// SIMATIC S7-200 project (STEP 7-Micro/WIN), CPU 224 REL 02.01

SYMBOL_TABLE USER1
lightSensor      V0.0
openDoor         V0.1
lowBob           V0.2
upBob            V0.3
heaterGoOn       V2.0
lightGoOn        V2.1
doorGoOpen       V2.2
ventilGoOn       V2.3
valve1goOn       V2.4
valve2goOn       V2.5
valve3goOn       V2.6
lightBySensor    V3.0
lightByTime      V3.1
lightHandOn      V3.2
lightHandOff     V3.3
heatSensorIsAir  V3.4
heatHandOn       V3.5
heatHandOff      V3.6
doorHandOn       V3.7
doorHandOff      V4.0
setClock         V4.1
readYear         VB50
readMonth        VB51
readDay          VB52
readHours        VB53
readMinutes      VB54
readSeconds      VB55
readWeekday      VB57
writeYear        VB58
writeMonth       VB59
writeDay         VB60
writeHours       VB61
writeMinutes     VB62
writeSeconds     VB63
writeWeekday     VB65
v1_e1_on_hh      VB148
v1_e1_on_mm      VB149
v1_e1_off_hh     VB150
v1_e1_off_mm     VB151
v1_e2_on_hh      VB152
v1_e2_on_mm      VB153
v1_e2_off_hh     VB154
v1_e2_off_mm     VB155
v1_e3_on_hh      VB156
v1_e3_on_mm      VB157
v1_e3_off_hh     VB158
v1_e3_off_mm     VB159
v1_e4_on_hh      VB160
v1_e4_on_mm      VB161
v1_e4_off_hh     VB162
v1_e4_off_mm     VB163
v1_e5_on_hh      VB164
v1_e5_on_mm      VB165
v1_e5_off_hh     VB166
v1_e5_off_mm     VB167
v2_e1_on_hh      VB168
v2_e1_on_mm      VB169
v2_e1_off_hh     VB170
v2_e1_off_mm     VB171
v2_e2_on_hh      VB172
v2_e2_on_mm      VB173
v2_e2_off_hh     VB174
v2_e2_off_mm     VB175
v2_e3_on_hh      VB176
v2_e3_on_mm      VB177
v2_e3_off_hh     VB178
v2_e3_off_mm     VB179
v2_e4_on_hh      VB180
v2_e4_on_mm      VB181
v2_e4_off_hh     VB182
v2_e4_off_mm     VB183
v2_e5_on_hh      VB184
v2_e5_on_mm      VB185
v2_e5_off_hh     VB186
v2_e5_off_mm     VB187
light_e1_on_hh   VB188
light_e1_on_mm   VB189
light_e1_off_hh  VB190
light_e1_off_mm  VB191
light_e2_on_hh   VB192
light_e2_on_mm   VB193
light_e2_off_hh  VB194
light_e2_off_mm  VB195
door_e1_on_hh    VB212
door_e1_on_mm    VB213
door_e1_off_hh   VB214
door_e1_off_mm   VB215
door_e2_on_hh    VB216
door_e2_on_mm    VB217
door_e2_off_hh   VB218
door_e2_off_mm   VB219
roomTemp4ma      VD100
roomTemp20ma     VD104
airTemp4ma       VD108
airTemp20ma      VD112
humidityRoom4ma  VD116
humidityRoom20ma VD120
floorTemp4ma     VD124
floorTemp20ma    VD128
roomTemp         VD132
airTemp          VD136
humidityRoom     VD140
floorTemp        VD144
lowSpWithAir     VD196
upSpWithAir      VD200
lowSpWithFloor   VD204
upSpWithFloor    VD208
lightTimeGo      V4.2
doorTimeGo       V4.3
heatTempGo       V4.4
lightHandGo      V4.5
doorHandGo       V4.6
heatHandGo       V4.7
ventilSensorIsTemp V5.0
lowSpWithTemp    VD220
upSpWithTemp     VD224
lowSpWithHumi    VD228
upSpWithHumi     VD232
lowSpWithOutside VD236
upSpWithOutside  VD240
heat2goOn        V5.1
im1_e1_on_hh     VB244
im1_e1_on_mm     VB245
im1_e1_off_hh    VB246
im1_e1_off_mm    VB247
im1_e2_on_hh     VB248
im1_e2_on_mm     VB249
im1_e2_off_hh    VB250
im1_e2_off_mm    VB251
im1_e3_on_hh     VB252
im1_e3_on_mm     VB253
im1_e3_off_hh    VB254
im1_e3_off_mm    VB255
im1_e4_on_hh     VB256
im1_e4_on_mm     VB257
im1_e4_off_hh    VB258
im1_e4_off_mm    VB259
im1_e5_on_hh     VB260
im1_e5_on_mm     VB261
im1_e5_off_hh    VB262
im1_e5_off_mm    VB263
im2_e1_on_hh     VB264
im2_e1_on_mm     VB265
im2_e1_off_hh    VB266
im2_e1_off_mm    VB267
im2_e2_on_hh     VB268
im2_e2_on_mm     VB269
im2_e2_off_hh    VB270
im2_e2_off_mm    VB271
im2_e3_on_hh     VB272
im2_e3_on_mm     VB273
im2_e3_off_hh    VB274
im2_e3_off_mm    VB275
im2_e4_on_hh     VB276
im2_e4_on_mm     VB277
im2_e4_off_hh    VB278
im2_e4_off_mm    VB279
im2_e5_on_hh     VB280
im2_e5_on_mm     VB281
im2_e5_off_hh    VB282
im2_e5_off_mm    VB283
im1goOn          V5.2
im2goOn          V5.3
END_SYMBOL_TABLE

ORGANIZATION_BLOCK Program_Block:OB1
TITLE=PROGRAM COMMENTS
BEGIN
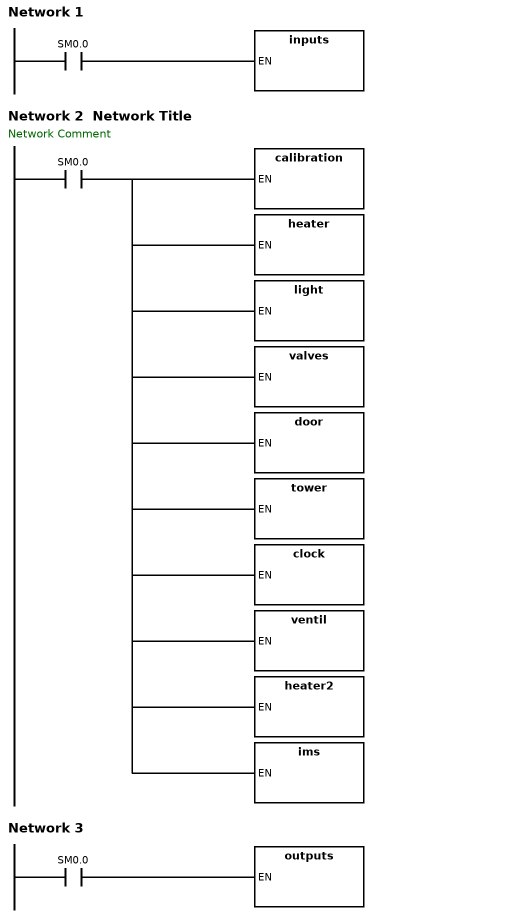
Network 1
LD     SM0.0
CALL   inputs:SBR3
Network 2 // Network Title
// Network Comment
LD     SM0.0
CALL   calibration:SBR0
CALL   heater:SBR6
CALL   light:SBR5
CALL   valves:SBR4
CALL   door:SBR7
CALL   tower:SBR9
CALL   clock:SBR2
CALL   ventil:SBR12
CALL   heater2:SBR13
CALL   ims:SBR14
Network 3
LD     SM0.0
CALL   outputs:SBR8
END_ORGANIZATION_BLOCK

SUBROUTINE_BLOCK calibration:SBR0
TITLE=SUBROUTINE COMMENTS
BEGIN
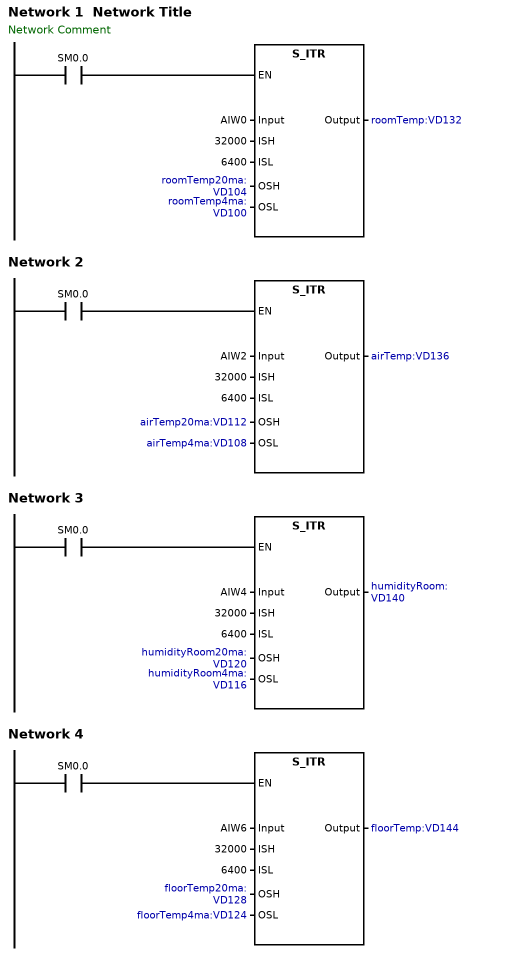
Network 1 // Network Title
// Network Comment
LD     SM0.0
CALL   S_ITR:SBR1, AIW0, 32000, 6400, roomTemp20ma:VD104, roomTemp4ma:VD100, roomTemp:VD132
Network 2
LD     SM0.0
CALL   S_ITR:SBR1, AIW2, 32000, 6400, airTemp20ma:VD112, airTemp4ma:VD108, airTemp:VD136
Network 3
LD     SM0.0
CALL   S_ITR:SBR1, AIW4, 32000, 6400, humidityRoom20ma:VD120, humidityRoom4ma:VD116, humidityRoom:VD140
Network 4
LD     SM0.0
CALL   S_ITR:SBR1, AIW6, 32000, 6400, floorTemp20ma:VD128, floorTemp4ma:VD124, floorTemp:VD144
END_SUBROUTINE_BLOCK

// SBR1: protected block, not included

SUBROUTINE_BLOCK clock:SBR2
TITLE=SUBROUTINE COMMENTS
BEGIN
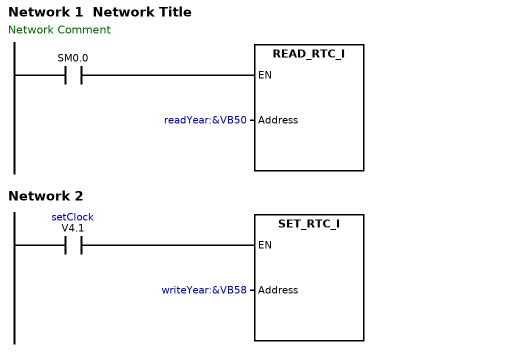
Network 1 // Network Title
// Network Comment
LD     SM0.0
CALL   READ_RTC_I:SBR10, &readYear:VB50
Network 2
LD     setClock:V4.1
CALL   SET_RTC_I:SBR11, &writeYear:VB58
END_SUBROUTINE_BLOCK

SUBROUTINE_BLOCK inputs:SBR3
TITLE=SUBROUTINE COMMENTS
BEGIN
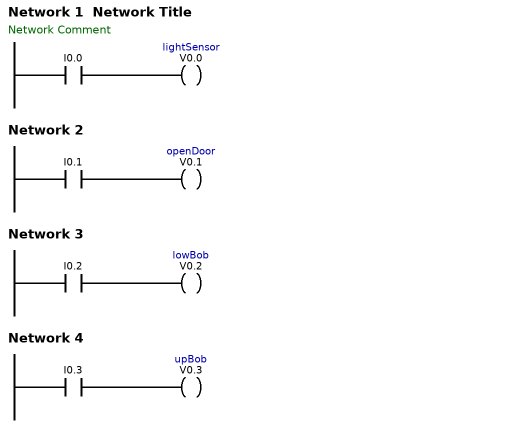
Network 1 // Network Title
// Network Comment
LD     I0.0
=      lightSensor:V0.0
Network 2
LD     I0.1
=      openDoor:V0.1
Network 3
LD     I0.2
=      lowBob:V0.2
Network 4
LD     I0.3
=      upBob:V0.3
END_SUBROUTINE_BLOCK

SUBROUTINE_BLOCK valves:SBR4
TITLE=SUBROUTINE COMMENTS
BEGIN
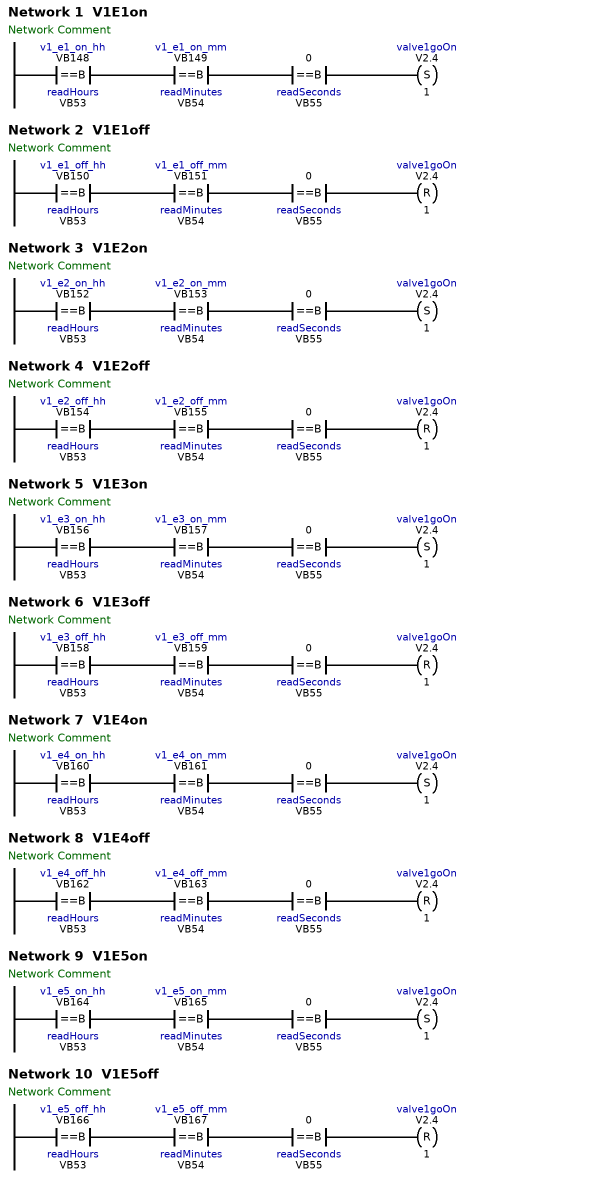
Network 1 // V1E1on
// Network Comment
LDB=   v1_e1_on_hh:VB148, readHours:VB53
AB=    v1_e1_on_mm:VB149, readMinutes:VB54
AB=    0, readSeconds:VB55
S      valve1goOn:V2.4, 1
Network 2 // V1E1off
// Network Comment
LDB=   v1_e1_off_hh:VB150, readHours:VB53
AB=    v1_e1_off_mm:VB151, readMinutes:VB54
AB=    0, readSeconds:VB55
R      valve1goOn:V2.4, 1
Network 3 // V1E2on
// Network Comment
LDB=   v1_e2_on_hh:VB152, readHours:VB53
AB=    v1_e2_on_mm:VB153, readMinutes:VB54
AB=    0, readSeconds:VB55
S      valve1goOn:V2.4, 1
Network 4 // V1E2off
// Network Comment
LDB=   v1_e2_off_hh:VB154, readHours:VB53
AB=    v1_e2_off_mm:VB155, readMinutes:VB54
AB=    0, readSeconds:VB55
R      valve1goOn:V2.4, 1
Network 5 // V1E3on
// Network Comment
LDB=   v1_e3_on_hh:VB156, readHours:VB53
AB=    v1_e3_on_mm:VB157, readMinutes:VB54
AB=    0, readSeconds:VB55
S      valve1goOn:V2.4, 1
Network 6 // V1E3off
// Network Comment
LDB=   v1_e3_off_hh:VB158, readHours:VB53
AB=    v1_e3_off_mm:VB159, readMinutes:VB54
AB=    0, readSeconds:VB55
R      valve1goOn:V2.4, 1
Network 7 // V1E4on
// Network Comment
LDB=   v1_e4_on_hh:VB160, readHours:VB53
AB=    v1_e4_on_mm:VB161, readMinutes:VB54
AB=    0, readSeconds:VB55
S      valve1goOn:V2.4, 1
Network 8 // V1E4off
// Network Comment
LDB=   v1_e4_off_hh:VB162, readHours:VB53
AB=    v1_e4_off_mm:VB163, readMinutes:VB54
AB=    0, readSeconds:VB55
R      valve1goOn:V2.4, 1
Network 9 // V1E5on
// Network Comment
LDB=   v1_e5_on_hh:VB164, readHours:VB53
AB=    v1_e5_on_mm:VB165, readMinutes:VB54
AB=    0, readSeconds:VB55
S      valve1goOn:V2.4, 1
Network 10 // V1E5off
// Network Comment
LDB=   v1_e5_off_hh:VB166, readHours:VB53
AB=    v1_e5_off_mm:VB167, readMinutes:VB54
AB=    0, readSeconds:VB55
R      valve1goOn:V2.4, 1
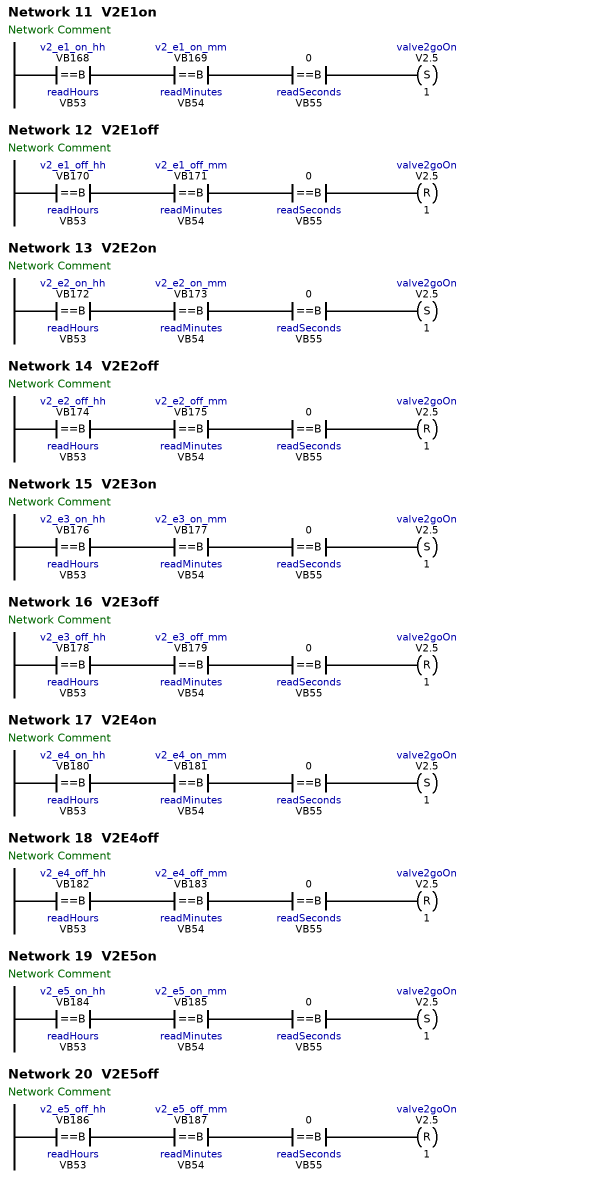
Network 11 // V2E1on
// Network Comment
LDB=   v2_e1_on_hh:VB168, readHours:VB53
AB=    v2_e1_on_mm:VB169, readMinutes:VB54
AB=    0, readSeconds:VB55
S      valve2goOn:V2.5, 1
Network 12 // V2E1off
// Network Comment
LDB=   v2_e1_off_hh:VB170, readHours:VB53
AB=    v2_e1_off_mm:VB171, readMinutes:VB54
AB=    0, readSeconds:VB55
R      valve2goOn:V2.5, 1
Network 13 // V2E2on
// Network Comment
LDB=   v2_e2_on_hh:VB172, readHours:VB53
AB=    v2_e2_on_mm:VB173, readMinutes:VB54
AB=    0, readSeconds:VB55
S      valve2goOn:V2.5, 1
Network 14 // V2E2off
// Network Comment
LDB=   v2_e2_off_hh:VB174, readHours:VB53
AB=    v2_e2_off_mm:VB175, readMinutes:VB54
AB=    0, readSeconds:VB55
R      valve2goOn:V2.5, 1
Network 15 // V2E3on
// Network Comment
LDB=   v2_e3_on_hh:VB176, readHours:VB53
AB=    v2_e3_on_mm:VB177, readMinutes:VB54
AB=    0, readSeconds:VB55
S      valve2goOn:V2.5, 1
Network 16 // V2E3off
// Network Comment
LDB=   v2_e3_off_hh:VB178, readHours:VB53
AB=    v2_e3_off_mm:VB179, readMinutes:VB54
AB=    0, readSeconds:VB55
R      valve2goOn:V2.5, 1
Network 17 // V2E4on
// Network Comment
LDB=   v2_e4_on_hh:VB180, readHours:VB53
AB=    v2_e4_on_mm:VB181, readMinutes:VB54
AB=    0, readSeconds:VB55
S      valve2goOn:V2.5, 1
Network 18 // V2E4off
// Network Comment
LDB=   v2_e4_off_hh:VB182, readHours:VB53
AB=    v2_e4_off_mm:VB183, readMinutes:VB54
AB=    0, readSeconds:VB55
R      valve2goOn:V2.5, 1
Network 19 // V2E5on
// Network Comment
LDB=   v2_e5_on_hh:VB184, readHours:VB53
AB=    v2_e5_on_mm:VB185, readMinutes:VB54
AB=    0, readSeconds:VB55
S      valve2goOn:V2.5, 1
Network 20 // V2E5off
// Network Comment
LDB=   v2_e5_off_hh:VB186, readHours:VB53
AB=    v2_e5_off_mm:VB187, readMinutes:VB54
AB=    0, readSeconds:VB55
R      valve2goOn:V2.5, 1
END_SUBROUTINE_BLOCK

SUBROUTINE_BLOCK light:SBR5
TITLE=SUBROUTINE COMMENTS
BEGIN
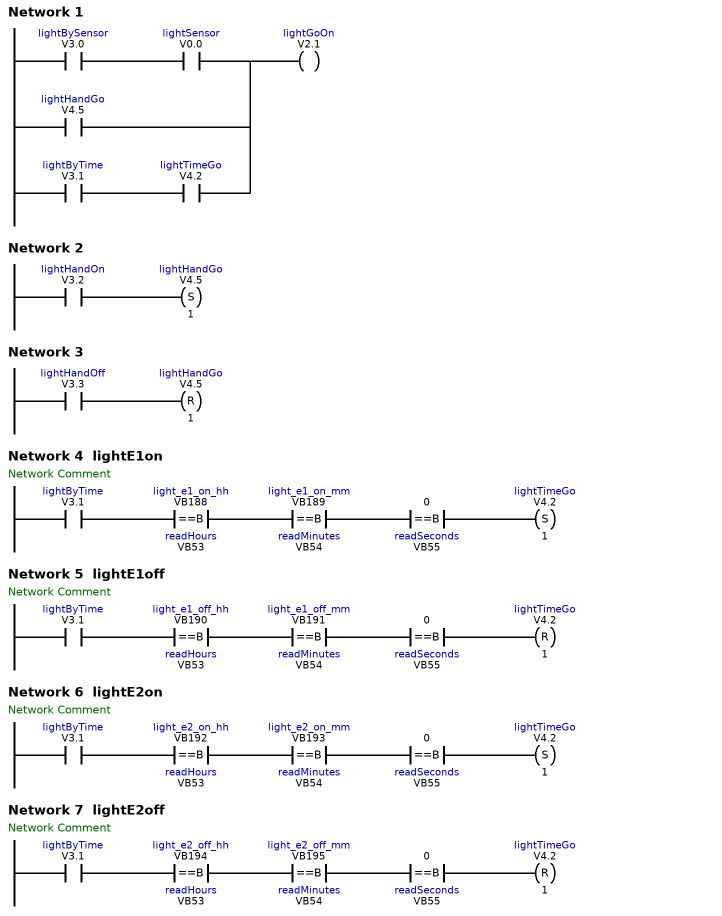
Network 1
LD     lightBySensor:V3.0
A      lightSensor:V0.0
O      lightHandGo:V4.5
LD     lightByTime:V3.1
A      lightTimeGo:V4.2
OLD
=      lightGoOn:V2.1
Network 2
LD     lightHandOn:V3.2
S      lightHandGo:V4.5, 1
Network 3
LD     lightHandOff:V3.3
R      lightHandGo:V4.5, 1
Network 4 // lightE1on
// Network Comment
LD     lightByTime:V3.1
AB=    light_e1_on_hh:VB188, readHours:VB53
AB=    light_e1_on_mm:VB189, readMinutes:VB54
AB=    0, readSeconds:VB55
S      lightTimeGo:V4.2, 1
Network 5 // lightE1off
// Network Comment
LD     lightByTime:V3.1
AB=    light_e1_off_hh:VB190, readHours:VB53
AB=    light_e1_off_mm:VB191, readMinutes:VB54
AB=    0, readSeconds:VB55
R      lightTimeGo:V4.2, 1
Network 6 // lightE2on
// Network Comment
LD     lightByTime:V3.1
AB=    light_e2_on_hh:VB192, readHours:VB53
AB=    light_e2_on_mm:VB193, readMinutes:VB54
AB=    0, readSeconds:VB55
S      lightTimeGo:V4.2, 1
Network 7 // lightE2off
// Network Comment
LD     lightByTime:V3.1
AB=    light_e2_off_hh:VB194, readHours:VB53
AB=    light_e2_off_mm:VB195, readMinutes:VB54
AB=    0, readSeconds:VB55
R      lightTimeGo:V4.2, 1
Network 8 // Network Title
// Network Comment
END_SUBROUTINE_BLOCK

SUBROUTINE_BLOCK heater:SBR6
TITLE=SUBROUTINE COMMENTS
BEGIN
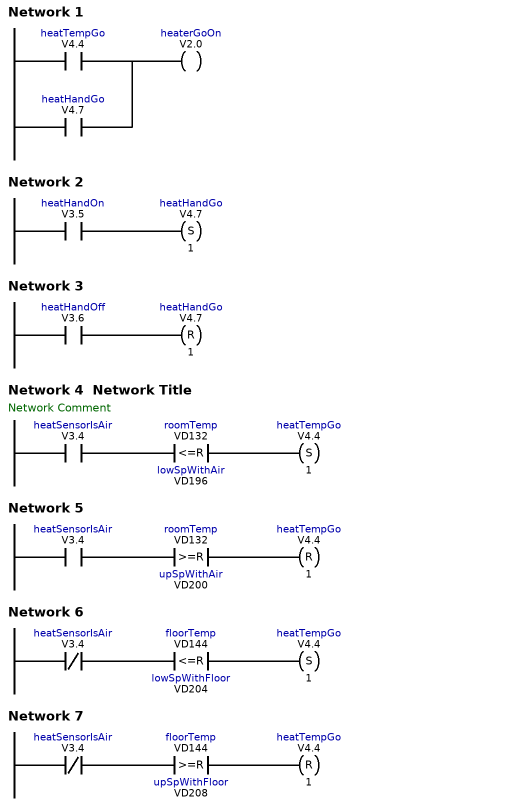
Network 1
LD     heatTempGo:V4.4
O      heatHandGo:V4.7
=      heaterGoOn:V2.0
Network 2
LD     heatHandOn:V3.5
S      heatHandGo:V4.7, 1
Network 3
LD     heatHandOff:V3.6
R      heatHandGo:V4.7, 1
Network 4 // Network Title
// Network Comment
LD     heatSensorIsAir:V3.4
AR<=   roomTemp:VD132, lowSpWithAir:VD196
S      heatTempGo:V4.4, 1
Network 5
LD     heatSensorIsAir:V3.4
AR>=   roomTemp:VD132, upSpWithAir:VD200
R      heatTempGo:V4.4, 1
Network 6
LDN    heatSensorIsAir:V3.4
AR<=   floorTemp:VD144, lowSpWithFloor:VD204
S      heatTempGo:V4.4, 1
Network 7
LDN    heatSensorIsAir:V3.4
AR>=   floorTemp:VD144, upSpWithFloor:VD208
R      heatTempGo:V4.4, 1
END_SUBROUTINE_BLOCK

SUBROUTINE_BLOCK door:SBR7
TITLE=SUBROUTINE COMMENTS
BEGIN
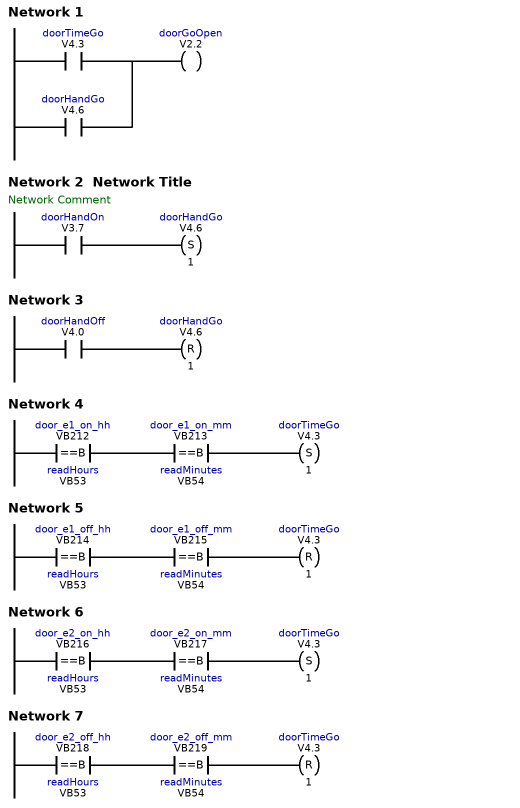
Network 1
LD     doorTimeGo:V4.3
O      doorHandGo:V4.6
=      doorGoOpen:V2.2
Network 2 // Network Title
// Network Comment
LD     doorHandOn:V3.7
S      doorHandGo:V4.6, 1
Network 3
LD     doorHandOff:V4.0
R      doorHandGo:V4.6, 1
Network 4
LDB=   door_e1_on_hh:VB212, readHours:VB53
AB=    door_e1_on_mm:VB213, readMinutes:VB54
S      doorTimeGo:V4.3, 1
Network 5
LDB=   door_e1_off_hh:VB214, readHours:VB53
AB=    door_e1_off_mm:VB215, readMinutes:VB54
R      doorTimeGo:V4.3, 1
Network 6
LDB=   door_e2_on_hh:VB216, readHours:VB53
AB=    door_e2_on_mm:VB217, readMinutes:VB54
S      doorTimeGo:V4.3, 1
Network 7
LDB=   door_e2_off_hh:VB218, readHours:VB53
AB=    door_e2_off_mm:VB219, readMinutes:VB54
R      doorTimeGo:V4.3, 1
END_SUBROUTINE_BLOCK

SUBROUTINE_BLOCK outputs:SBR8
TITLE=SUBROUTINE COMMENTS
BEGIN
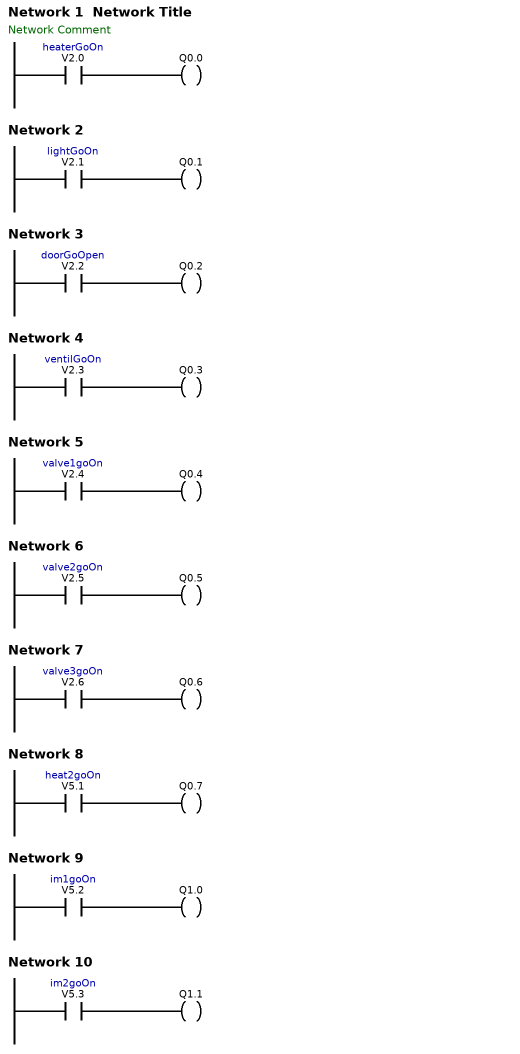
Network 1 // Network Title
// Network Comment
LD     heaterGoOn:V2.0
=      Q0.0
Network 2
LD     lightGoOn:V2.1
=      Q0.1
Network 3
LD     doorGoOpen:V2.2
=      Q0.2
Network 4
LD     ventilGoOn:V2.3
=      Q0.3
Network 5
LD     valve1goOn:V2.4
=      Q0.4
Network 6
LD     valve2goOn:V2.5
=      Q0.5
Network 7
LD     valve3goOn:V2.6
=      Q0.6
Network 8
LD     heat2goOn:V5.1
=      Q0.7
Network 9
LD     im1goOn:V5.2
=      Q1.0
Network 10
LD     im2goOn:V5.3
=      Q1.1
END_SUBROUTINE_BLOCK

SUBROUTINE_BLOCK tower:SBR9
TITLE=SUBROUTINE COMMENTS
BEGIN
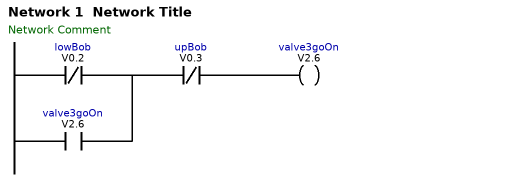
Network 1 // Network Title
// Network Comment
LDN    lowBob:V0.2
O      valve3goOn:V2.6
AN     upBob:V0.3
=      valve3goOn:V2.6
END_SUBROUTINE_BLOCK

// SBR10: protected block, not included

// SBR11: protected block, not included

SUBROUTINE_BLOCK ventil:SBR12
TITLE=
BEGIN
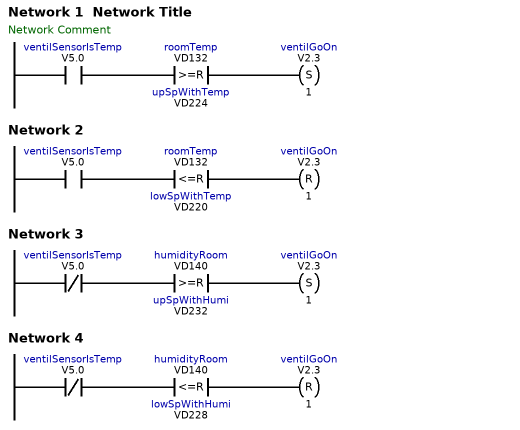
Network 1 // Network Title
// Network Comment
LD     ventilSensorIsTemp:V5.0
AR>=   roomTemp:VD132, upSpWithTemp:VD224
S      ventilGoOn:V2.3, 1
Network 2
LD     ventilSensorIsTemp:V5.0
AR<=   roomTemp:VD132, lowSpWithTemp:VD220
R      ventilGoOn:V2.3, 1
Network 3
LDN    ventilSensorIsTemp:V5.0
AR>=   humidityRoom:VD140, upSpWithHumi:VD232
S      ventilGoOn:V2.3, 1
Network 4
LDN    ventilSensorIsTemp:V5.0
AR<=   humidityRoom:VD140, lowSpWithHumi:VD228
R      ventilGoOn:V2.3, 1
END_SUBROUTINE_BLOCK

SUBROUTINE_BLOCK heater2:SBR13
TITLE=
BEGIN
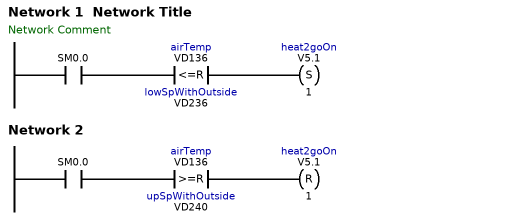
Network 1 // Network Title
// Network Comment
// (network saved uncompiled; LAD cells follow)
// row 0: c0 -| |- SM0.0  c1 -|<=R|- airTemp:VD136, lowSpWithOutside:VD236  c2 -(S) heat2goOn:V5.1, 1
Network 2
// (network saved uncompiled; LAD cells follow)
// row 0: c0 -| |- SM0.0  c1 -|>=R|- airTemp:VD136, upSpWithOutside:VD240  c2 -(R) heat2goOn:V5.1, 1
END_SUBROUTINE_BLOCK

SUBROUTINE_BLOCK ims:SBR14
TITLE=
BEGIN
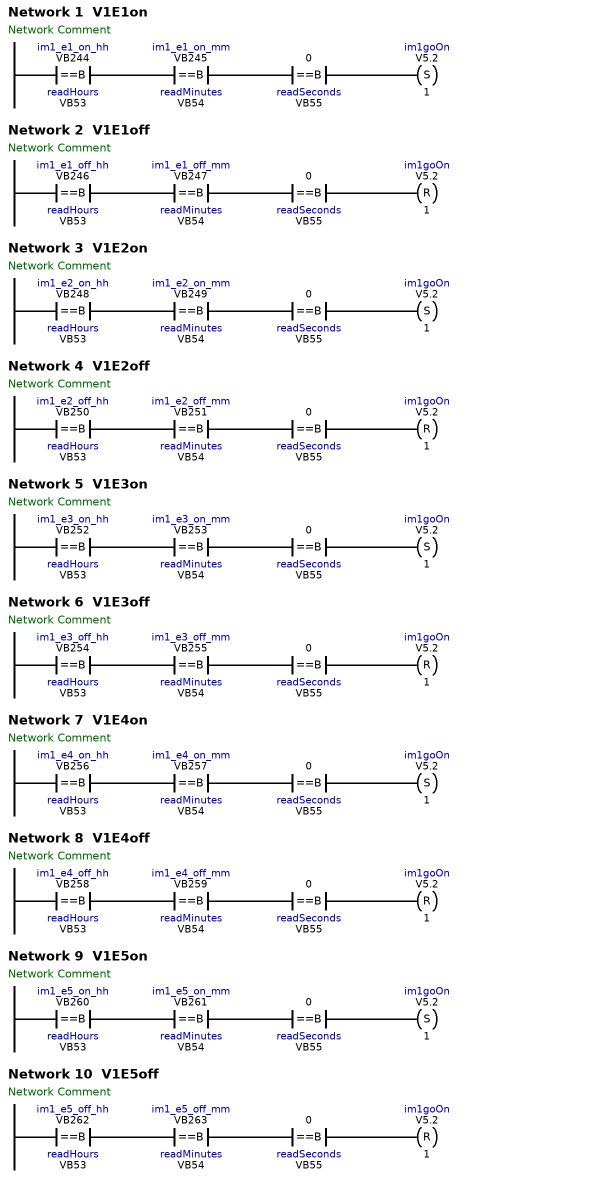
Network 1 // V1E1on
// Network Comment
LDB=   im1_e1_on_hh:VB244, readHours:VB53
AB=    im1_e1_on_mm:VB245, readMinutes:VB54
AB=    0, readSeconds:VB55
S      im1goOn:V5.2, 1
Network 2 // V1E1off
// Network Comment
LDB=   im1_e1_off_hh:VB246, readHours:VB53
AB=    im1_e1_off_mm:VB247, readMinutes:VB54
AB=    0, readSeconds:VB55
R      im1goOn:V5.2, 1
Network 3 // V1E2on
// Network Comment
LDB=   im1_e2_on_hh:VB248, readHours:VB53
AB=    im1_e2_on_mm:VB249, readMinutes:VB54
AB=    0, readSeconds:VB55
S      im1goOn:V5.2, 1
Network 4 // V1E2off
// Network Comment
LDB=   im1_e2_off_hh:VB250, readHours:VB53
AB=    im1_e2_off_mm:VB251, readMinutes:VB54
AB=    0, readSeconds:VB55
R      im1goOn:V5.2, 1
Network 5 // V1E3on
// Network Comment
LDB=   im1_e3_on_hh:VB252, readHours:VB53
AB=    im1_e3_on_mm:VB253, readMinutes:VB54
AB=    0, readSeconds:VB55
S      im1goOn:V5.2, 1
Network 6 // V1E3off
// Network Comment
LDB=   im1_e3_off_hh:VB254, readHours:VB53
AB=    im1_e3_off_mm:VB255, readMinutes:VB54
AB=    0, readSeconds:VB55
R      im1goOn:V5.2, 1
Network 7 // V1E4on
// Network Comment
LDB=   im1_e4_on_hh:VB256, readHours:VB53
AB=    im1_e4_on_mm:VB257, readMinutes:VB54
AB=    0, readSeconds:VB55
S      im1goOn:V5.2, 1
Network 8 // V1E4off
// Network Comment
LDB=   im1_e4_off_hh:VB258, readHours:VB53
AB=    im1_e4_off_mm:VB259, readMinutes:VB54
AB=    0, readSeconds:VB55
R      im1goOn:V5.2, 1
Network 9 // V1E5on
// Network Comment
LDB=   im1_e5_on_hh:VB260, readHours:VB53
AB=    im1_e5_on_mm:VB261, readMinutes:VB54
AB=    0, readSeconds:VB55
S      im1goOn:V5.2, 1
Network 10 // V1E5off
// Network Comment
LDB=   im1_e5_off_hh:VB262, readHours:VB53
AB=    im1_e5_off_mm:VB263, readMinutes:VB54
AB=    0, readSeconds:VB55
R      im1goOn:V5.2, 1
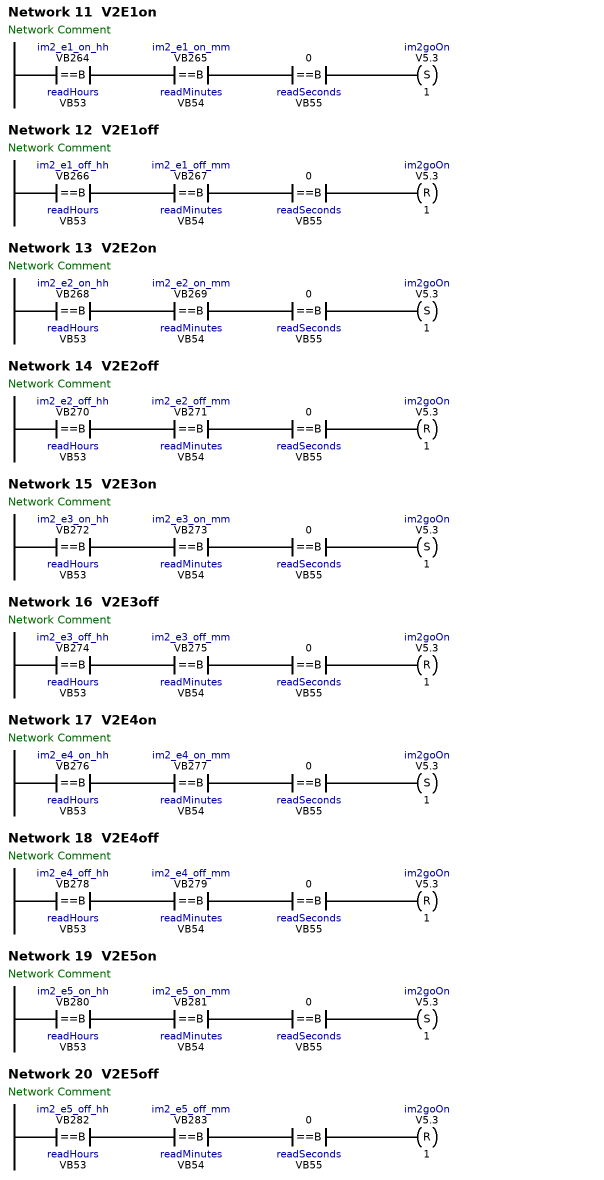
Network 11 // V2E1on
// Network Comment
LDB=   im2_e1_on_hh:VB264, readHours:VB53
AB=    im2_e1_on_mm:VB265, readMinutes:VB54
AB=    0, readSeconds:VB55
S      im2goOn:V5.3, 1
Network 12 // V2E1off
// Network Comment
LDB=   im2_e1_off_hh:VB266, readHours:VB53
AB=    im2_e1_off_mm:VB267, readMinutes:VB54
AB=    0, readSeconds:VB55
R      im2goOn:V5.3, 1
Network 13 // V2E2on
// Network Comment
LDB=   im2_e2_on_hh:VB268, readHours:VB53
AB=    im2_e2_on_mm:VB269, readMinutes:VB54
AB=    0, readSeconds:VB55
S      im2goOn:V5.3, 1
Network 14 // V2E2off
// Network Comment
LDB=   im2_e2_off_hh:VB270, readHours:VB53
AB=    im2_e2_off_mm:VB271, readMinutes:VB54
AB=    0, readSeconds:VB55
R      im2goOn:V5.3, 1
Network 15 // V2E3on
// Network Comment
LDB=   im2_e3_on_hh:VB272, readHours:VB53
AB=    im2_e3_on_mm:VB273, readMinutes:VB54
AB=    0, readSeconds:VB55
S      im2goOn:V5.3, 1
Network 16 // V2E3off
// Network Comment
LDB=   im2_e3_off_hh:VB274, readHours:VB53
AB=    im2_e3_off_mm:VB275, readMinutes:VB54
AB=    0, readSeconds:VB55
R      im2goOn:V5.3, 1
Network 17 // V2E4on
// Network Comment
LDB=   im2_e4_on_hh:VB276, readHours:VB53
AB=    im2_e4_on_mm:VB277, readMinutes:VB54
AB=    0, readSeconds:VB55
S      im2goOn:V5.3, 1
Network 18 // V2E4off
// Network Comment
LDB=   im2_e4_off_hh:VB278, readHours:VB53
AB=    im2_e4_off_mm:VB279, readMinutes:VB54
AB=    0, readSeconds:VB55
R      im2goOn:V5.3, 1
Network 19 // V2E5on
// Network Comment
LDB=   im2_e5_on_hh:VB280, readHours:VB53
AB=    im2_e5_on_mm:VB281, readMinutes:VB54
AB=    0, readSeconds:VB55
S      im2goOn:V5.3, 1
Network 20 // V2E5off
// Network Comment
LDB=   im2_e5_off_hh:VB282, readHours:VB53
AB=    im2_e5_off_mm:VB283, readMinutes:VB54
AB=    0, readSeconds:VB55
R      im2goOn:V5.3, 1
END_SUBROUTINE_BLOCK
